SUBAPPLICATION mapping_AuxFunction2_IX (* Mapping for all AuxFunction2 *)
  (* Standard: 61499-2 *)
  (* Version 1.0, 2023-01-29, Franz *)
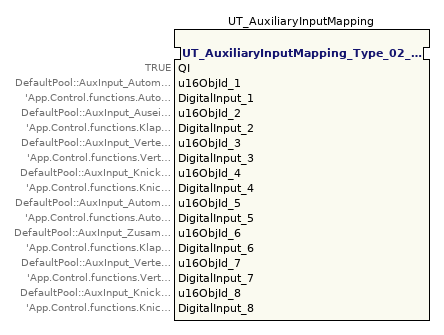
  FBS
    UT_AuxiliaryInputMapping : UT_AuxiliaryInputMapping_Type_02_Bool_NonLatched(QI := TRUE, u16ObjId_1 := DefaultPool::AuxInput_Automatik_ein, DigitalInput_1 := 'App.Control.functions.Automatik.ein.AuxInput', u16ObjId_2 := DefaultPool::AuxInput_Auseinanderklappen, DigitalInput_2 := 'App.Control.functions.Klappen.AuxInput_heben.IX', u16ObjId_3 := DefaultPool::AuxInput_Verteiler_senken, DigitalInput_3 := 'App.Control.functions.Verteiler.AuxInput_senken.IX', u16ObjId_4 := DefaultPool::AuxInput_Knickdeichsel_senken, DigitalInput_4 := 'App.Control.functions.Knickdeichsel.AuxInput_senken.IX', u16ObjId_5 := DefaultPool::AuxInput_Automatik_aus, DigitalInput_5 := 'App.Control.functions.Automatik.aus.AuxInput', u16ObjId_6 := DefaultPool::AuxInput_Zusammenklappen, DigitalInput_6 := 'App.Control.functions.Klappen.AuxInput_senken.IX', u16ObjId_7 := DefaultPool::AuxInput_Verteiler_heben, DigitalInput_7 := 'App.Control.functions.Verteiler.AuxInput_heben.IX', u16ObjId_8 := DefaultPool::AuxInput_Knickdeichsel_heben, DigitalInput_8 := 'App.Control.functions.Knickdeichsel.AuxInput_heben.IX');
  END_FBS
END_SUBAPPLICATION
